TYPE "Prod_CIn"
VERSION : 0.1
// Block: Prod_CIn
   STRUCT
      Rst : Bool;
      Part_Execution : Prod_Part_Done;
      Part_Prod : Prod_Part_Area;
      Beam_Prod : Prod_Beam_Area;
      Coil_Prod : Prod_Coil_Area;
   END_STRUCT;

END_TYPE
